(* LS Electric XG5000 project: BURNER110526 *)
(* PLC LSPLC *)
(* module base 0 slot 0: FEnet:XGL-EFMT(B) (Fast Ethernet Module, Electrical Master) *)
(* module base 0 slot 1: Cnet:XGL-C42A/B (Cnet Module(RS-422/485, RS-422/485)) *)
(* module base 0 slot 2: Input Module:XGI-D24A/B (DC 24V Input, 32 Contacts) *)
(* module base 0 slot 3: Input Module:XGI-D24A/B (DC 24V Input, 32 Contacts) *)
(* module base 0 slot 4: Output Module:XGQ-RY2A/B (Relay Output, 16 Contacts (2A, No Varistor/Varistor)) *)
(* module base 0 slot 5: Output Module:XGQ-RY2A/B (Relay Output, 16 Contacts (2A, No Varistor/Varistor)) *)
(* module base 0 slot 6: Analog Output Module:XGF-DC4S (Isolated-type Current Output Type(4 Channels)) *)
(* module base 0 slot 7: Analog Input Module:XGF-AD8A (A/D Voltage/Current Input Type(8 Channels)) *)
(* module base 0 slot 8: Temp. Measuring Module:XGF-RD4A (Temperature Input Type(4 Channels)) *)
VAR_GLOBAL
    GIA_TRI_SV : BOOL;
    _0006_CH0_DATA AT %UW0.6.3 : INT; (* Analog Output Module: CH0 Input *)
    _0006_CH0_OUTEN AT %UX0.6.32 : BOOL; (* Analog Output Module: CH0 Output Enable *)
    _0006_CH1_DATA AT %UW0.6.4 : INT; (* Analog Output Module: CH1 Input *)
    _0006_CH1_OUTEN AT %UX0.6.33 : BOOL; (* Analog Output Module: CH1 Output Enable *)
    _0006_CH2_DATA AT %UW0.6.5 : INT; (* Analog Output Module: CH2 Input *)
    _0006_CH2_OUTEN AT %UX0.6.34 : BOOL; (* Analog Output Module: CH2 Output Enable *)
    _0007_CH0_ACT AT %UX0.7.16 : BOOL; (* Analog Input Module: CH0 Activation Status *)
    _0007_CH0_DATA AT %UW0.7.2 : INT; (* Analog Input Module: CH0 Output *)
    _0007_CH1_ACT AT %UX0.7.17 : BOOL; (* Analog Input Module: CH1 Activation Status *)
    _0007_CH1_DATA AT %UW0.7.3 : INT; (* Analog Input Module: CH1 Output *)
    _0008_CH0_ACT AT %UX0.8.16 : BOOL; (* Temp. Measuring Module: CH0 Activation Status *)
    _0008_CH0_TEMP AT %UW0.8.4 : INT; (* Temp. Measuring Module: CH0 Temp. Data *)
END_VAR

(* Comments on direct variables
%MX98	Burner_Doul
%MX186	HMI_REMOTE
%MX187	HMI_LOCAL
%MX188	HMI_TEX_REMOTE
%MX189	HMI_TEX_LOCAL
%MX192	HMI_REMOTTE
%MX193	HMO_LOACAL
%MW15	DATA_MV_GZ900_ESV
%MW16	DATA_PV_GZ900_ESV
%MW17	DATA_SV_GZ900_ESV
%MW18	DATA_OVER_HTP_ESV
*)

PROGRAM NewProgram (* task: Scan Program *)
VAR
    AIR_CHECK : BOOL;
    AIR_CHECK_OK : BOOL;
    ALARM_AIR_SPEDD : BOOL;
    Alarm_ESV AT %MW5.8 : BOOL;
    ALARM_HIGHT_TEMP : BOOL;
    ALARM_MISS_FIRE : BOOL;
    ALARM_NO1_SHUT : BOOL;
    ALARM_NO2_SHUT : BOOL;
    ALARM_PRESS : BOOL;
    ALARM_SEVOR_HIG : BOOL;
    ALARM_SEVOR_LOW : BOOL;
    BUNER_START : BOOL;
    Burner_Doul AT %MX98 : BOOL;
    burner_Sing AT %MW6.1 : BOOL;
    BUR_START_PER AT %MW1.5 : BOOL; (* BURNER START PERMISSIVE *)
    B_EMG_STOP AT %MW0.0 : BOOL; (* EMEGENCY STOP *)
    B_RESET AT %MW0.1 : BOOL; (* BUTTON RESET *)
    checkk : BOOL;
    CHECK_HIG_SEVOR_OK : BOOL;
    CHECK_NO1_SHUT_OK : BOOL;
    CHECK_NO2_SHUT_OK : BOOL;
    Circulation_Low_Speed_ESV AT %MW5.2 : BOOL;
    Combustion_Air_Fan_Fault_ESV AT %MW4.13 : BOOL;
    Combustion_Air_Fan_Run_ESV AT %MW4.2 : BOOL;
    ECOR_TRIP : BOOL;
    Emergency_Stop_ESV AT %MW5.1 : BOOL;
    FAN_RUN AT %MW0.6 : BOOL; (* LOW CIRCULATION FAN SPEED *)
    FLAMON : BOOL;
    Gas_Leak_Check_Switch_Fault_ESV AT %MW5.4 : BOOL;
    Gas_Leak_PSH_ESV AT %MW4.5 : BOOL;
    Gas_Leak_PSL_ESV AT %MW5.0 : BOOL;
    Gas_Pressure_Hi_ESV AT %MW4.8 : BOOL;
    Gas_Pressure_Low_ESV AT %MW5.3 : BOOL;
    HIGH_GAS_LEAK_PRE AT %MW1.11 : BOOL; (* HIGH GAS LEAK PRESSURE CONTROL SWITCH *)
    HIGH_GAS_PRE AT %MW1.8 : BOOL; (* HIGH GAS PRESSURE *)
    HIGH_LIMIT : BOOL;
    HIGH_SEVOR_CHECK : BOOL;
    Hi_Fire_Limit_Switch_ESV AT %MW4.3 : BOOL;
    Hi_Fire_Limit_Switch_Fault_ESV AT %MW4.12 : BOOL;
    HMI : BOOL;
    HPV_Temp AT %MW507 : INT;
    HPV_Temp1 AT %MW508 : INT;
    INST : TON;
    INST1 : TON;
    INST10 : TON;
    INST11 : TON;
    INST12 : TON;
    INST13 : TON;
    INST14 : TON;
    INST15 : TON;
    INST16 : TON;
    INST17 : TON;
    INST18 : TON;
    INST19 : TON;
    INST2 : TON;
    INST20 : TON;
    INST21 : TON;
    INST22 : TON;
    INST23 : TON;
    INST24 : CTU_INT;
    INST25 : TON;
    INST26 : TON;
    INST27 : TON;
    INST28 : TON;
    INST29 : TON;
    INST3 : TON;
    INST30 : TON;
    INST4 : TON;
    INST5 : TON;
    INST6 : TON;
    INST7 : TON;
    INST8 : TON;
    INST9 : TON;
    LOW_AIR_PRE : BOOL;
    Low_Comb_Air_Fan_Pr_ESV AT %MW4.9 : BOOL;
    LOW_FIRE : BOOL;
    LOW_GAS_LEAK_PRE AT %MW1.10 : BOOL; (* LOW GAS LEAK PRESSURE CONTROL SWITCH *)
    LOW_GAS_PRE AT %MW1.7 : BOOL; (* LOW GAS PRESSURE *)
    LOW_LIMIT : BOOL;
    LOW_LIMIT_CHECK_OK : BOOL;
    Lo_Fire_Limit_Switch_ESV AT %MW4.14 : BOOL;
    Lo_Fire_Limit_Switch_Fault_ESV AT %MW5.7 : BOOL;
    Main_Burner_Miss_Fire_ESV AT %MW5.6 : BOOL;
    MAIN_BURNER_START : BOOL;
    Main_Gas_Shutoff_ESV AT %MW4.15 : BOOL;
    MAIN_PANEL_READY : BOOL;
    Man_Auto_GZ900 AT %MW101 : INT;
    Man_MV_GZ900 AT %MW100 : INT;
    MG : BOOL;
    MG1 AT %MW0.4 : BOOL; (* #1  COMBUSTION FAN RUN *)
    MG2 AT %MW0.5 : BOOL; (* #2  COMBUSTION FAN RUN *)
    MV_GZ900_OUT : INT;
    MƯ20 : WORD;
    mư4 : WORD;
    NO1_ECOR_TRIP AT %MW0.2 : BOOL; (* #1 FAN ECOR TRIP *)
    NO1_FLAME_ON AT %MW1.14 : BOOL; (* #1 BURNER FLAME ON SIGNAL *)
    NO1_HIGH_LIMIT AT %MW1.1 : BOOL; (* #1 HIGH FIRE LIMIT SWITCH *)
    NO1_LOW_AIR_PRE AT %MW1.9 : BOOL; (* #1 LOW COMBUSTION AIR PRESSURE *)
    NO1_LOW_LIMIT AT %MW1.0 : BOOL; (* #1 LOW FIRE LIMIT SWITCH *)
    NO1_SHUT_CHECK : BOOL;
    NO1_SHUT_OFF_SW AT %MW1.13 : BOOL; (* #1 MAIN SHUT_OFF VAVLE CLOSED LIMIT SWITCH *)
    NO2_ECOR_TRIP AT %MW0.3 : BOOL; (* #2 FAN ECOR TRIP *)
    NO2_FLAME_ON AT %MW1.15 : BOOL; (* #2 BURNER FLAME ON SIGNAL *)
    NO2_HIGH_LIMIT AT %MW1.3 : BOOL; (* #2 HIGH FIRE LIMIT SWITCH *)
    NO2_LOW_AIR_PRE AT %MW1.12 : BOOL; (* #2 LOW COMBUSTION AIR PRESSURE *)
    NO2_LOW_LIMIT AT %MW1.2 : BOOL; (* #2 LOW FIRE LIMIT SWITCH *)
    NO2_SHUT_CHECK : BOOL;
    NO_READY : BOOL;
    O502 AT %MW3.0 : BOOL; (* BURNER LOAD UP *)
    O503 AT %MW3.1 : BOOL; (* LOW CIRCULATION FAN SPEED *)
    O504 AT %MW3.2 : BOOL; (* BURNER START *)
    O505 AT %MW3.3 : BOOL;
    O506 AT %MW3.4 : BOOL; (* HIGH TEMPERATURE *)
    O507 AT %MW3.5 : BOOL; (* MISS FIRE *)
    O508 AT %MW3.6 : BOOL; (* HIGH GAS PRESSURE *)
    O509 AT %MW3.7 : BOOL; (* LOW GAS PRESSURE *)
    O510 AT %MW3.8 : BOOL; (* GAS LEAK FAULT *)
    O511 AT %MW3.9 : BOOL; (* PURGE START *)
    O512 AT %MW3.10 : BOOL; (* PURGE END *)
    O513 AT %MW3.11 : BOOL; (* NO 1 LOW COMBUSTION FAN PRESSURE *)
    O514 AT %MW3.12 : BOOL; (* NO 1 LOW COMBUSTION FAN RUNNING *)
    O515 AT %MW3.13 : BOOL; (* NO 2 LOW COMBUSTION FAN PRESSURE *)
    O516 AT %MW3.14 : BOOL; (* NO 2 LOW COMBUSTION FAN RUNNING *)
    O517 AT %MW3.15 : BOOL;
    O518 AT %MW2.14 : BOOL; (* NO.01 COMBUSTION FAN ECOR TRIP *)
    O519 AT %MW2.15 : BOOL; (* NO.02 COMBUSTION FAN ECOR TRIP *)
    Operation_Remote_Mode_ESV AT %MW4.6 : BOOL;
    Pilot_Burner_Miss_Fire_ESV AT %MW4.11 : BOOL;
    PILOT_INR : BOOL;
    Pilot_Valve_ESV AT %MW4.4 : BOOL;
    PV_GZ900 AT %MW103 : INT;
    PV_GZ900_OUT : INT;
    Ready_ESV AT %MW4.0 : BOOL;
    Remote_ESV AT %MW4.1 : BOOL;
    RE_RESET AT %MW1.6 : BOOL; (* REMOTE RESET *)
    RE_START AT %MW1.4 : BOOL; (* REMOTE START *)
    RMV_GZ900 AT %MW104 : INT;
    START : BOOL;
    STOP AT %MW6.0 : BOOL;
    STOP_BURNER : BOOL;
    SV_GZ900 AT %MW102 : INT;
    SV_THIC_Data AT %MW506 : INT;
    SV_TIC_Data AT %MW505 : INT;
    temp1 : INT;
    temp2 : INT;
    Temp_high_ESV AT %MW4.7 : BOOL;
    WMV_GZ900 AT %MW504 : INT;
    WPV AT %MW520 : INT;
    WPV_GZ900 AT %MW503 : INT;
    _1ST_Valve_Gas_leak_ESV AT %MW4.10 : BOOL;
    _2ND_Valve_Gas_leak_ESV AT %MW5.5 : BOOL;
END_VAR
VAR_EXTERNAL
    _0006_CH0_DATA : INT; (* AT %UW0.6.3 *) (* Analog Output Module: CH0 Input *)
    _0006_CH0_OUTEN : BOOL; (* AT %UX0.6.32 *) (* Analog Output Module: CH0 Output Enable *)
    _0006_CH1_DATA : INT; (* AT %UW0.6.4 *) (* Analog Output Module: CH1 Input *)
    _0006_CH1_OUTEN : BOOL; (* AT %UX0.6.33 *) (* Analog Output Module: CH1 Output Enable *)
    _0006_CH2_DATA : INT; (* AT %UW0.6.5 *) (* Analog Output Module: CH2 Input *)
    _0006_CH2_OUTEN : BOOL; (* AT %UX0.6.34 *) (* Analog Output Module: CH2 Output Enable *)
    _0007_CH0_ACT : BOOL; (* AT %UX0.7.16 *) (* Analog Input Module: CH0 Activation Status *)
    _0007_CH0_DATA : INT; (* AT %UW0.7.2 *) (* Analog Input Module: CH0 Output *)
    _0007_CH1_ACT : BOOL; (* AT %UX0.7.17 *) (* Analog Input Module: CH1 Activation Status *)
    _0007_CH1_DATA : INT; (* AT %UW0.7.3 *) (* Analog Input Module: CH1 Output *)
    _0008_CH0_ACT : BOOL; (* AT %UX0.8.16 *) (* Temp. Measuring Module: CH0 Activation Status *)
    _0008_CH0_TEMP : INT; (* AT %UW0.8.4 *) (* Temp. Measuring Module: CH0 Temp. Data *)
END_VAR
VAR
    _e1 : R_TRIG;
    _e2 : R_TRIG;
    _e3 : F_TRIG;
    _e4 : R_TRIG;
    _e5 : R_TRIG;
    _p6 : BOOL;
    _p7 : BOOL;
    _e8 : R_TRIG;
    _e9 : R_TRIG;
    _p10 : BOOL;
    _p11 : BOOL;
    _p12 : BOOL;
    _p13 : BOOL;
    _p14 : BOOL;
    _p15 : BOOL;
    _p16 : BOOL;
    _p17 : BOOL;
    _p18 : BOOL;
    _t19 : BOOL;
    _t20 : BOOL;
END_VAR

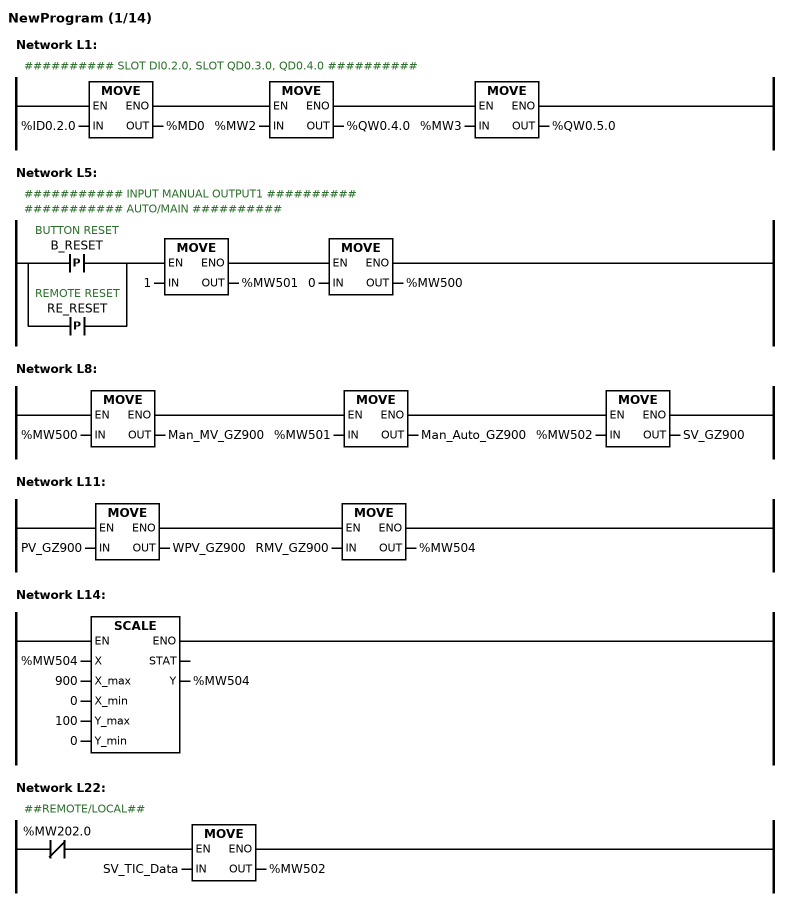
(* ########## SLOT DI0.2.0, SLOT QD0.3.0, QD0.4.0 ########## *)
(* Rung L1 *)
%MD0 := %ID0.2.0;
%QW0.4.0 := %MW2;
%QW0.5.0 := %MW3;
(* ########### INPUT MANUAL OUTPUT1 ########## / ########### AUTO/MAIN ########## *)
(* Rung L5 *)
_e1(CLK := B_RESET);
_e2(CLK := RE_RESET);
IF _e1.Q OR _e2.Q THEN
    %MW501 := 1;
    %MW500 := 0;
END_IF;
(* Rung L8 *)
Man_MV_GZ900 := %MW500;
Man_Auto_GZ900 := %MW501;
SV_GZ900 := %MW502;
(* Rung L11 *)
WPV_GZ900 := PV_GZ900;
%MW504 := RMV_GZ900;
(* Rung L14 *)
SCALE(X := %MW504, X_max := 900, X_min := 0, Y_max := 100, Y_min := 0, Y => %MW504);
(* ##REMOTE/LOCAL## *)
(* Rung L22 *)
IF NOT %MW202.0 THEN %MW502 := SV_TIC_Data; END_IF;

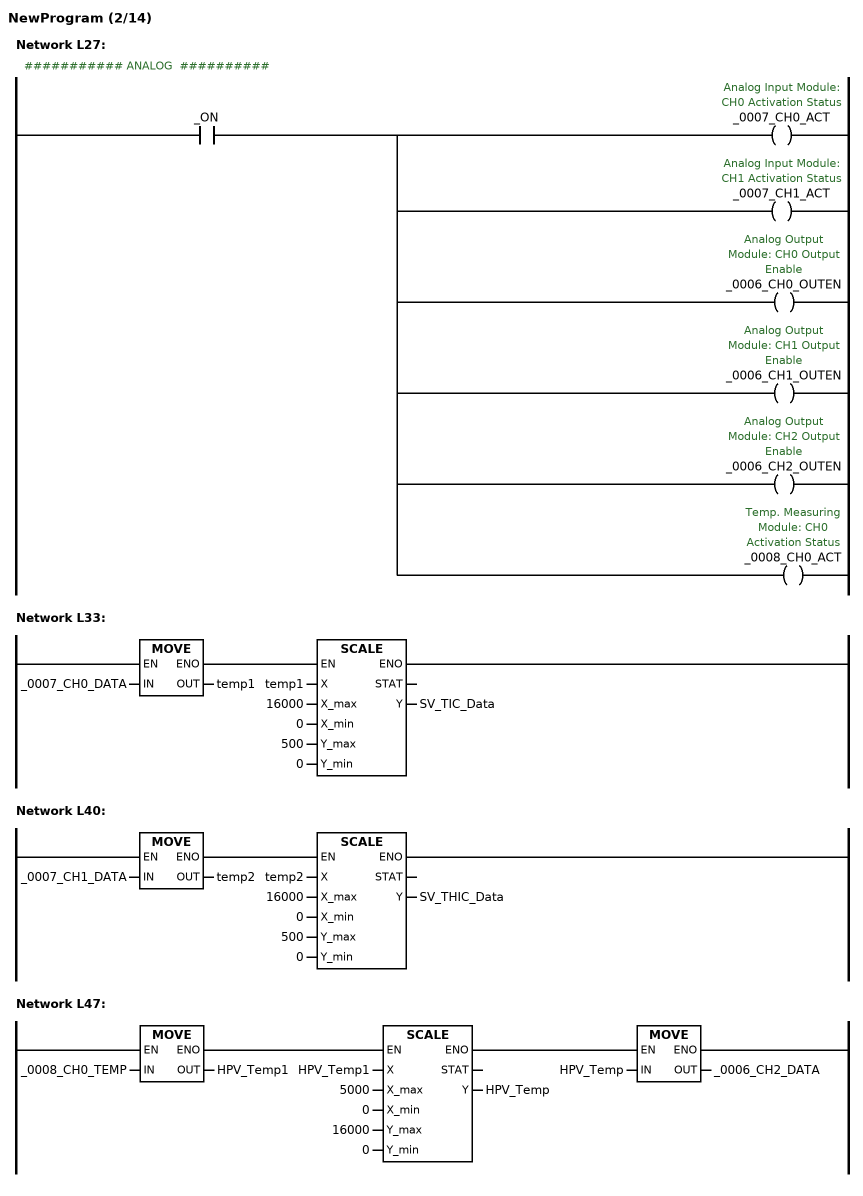
(* ########### ANALOG  ########## *)
(* Rung L27 *)
_0007_CH0_ACT := _ON;
_0007_CH1_ACT := _ON;
_0006_CH0_OUTEN := _ON;
_0006_CH1_OUTEN := _ON;
_0006_CH2_OUTEN := _ON;
_0008_CH0_ACT := _ON;
(* Rung L33 *)
temp1 := _0007_CH0_DATA;
SCALE(X := temp1, X_max := 16000, X_min := 0, Y_max := 500, Y_min := 0, Y => SV_TIC_Data);
(* Rung L40 *)
temp2 := _0007_CH1_DATA;
SCALE(X := temp2, X_max := 16000, X_min := 0, Y_max := 500, Y_min := 0, Y => SV_THIC_Data);
(* Rung L47 *)
HPV_Temp1 := _0008_CH0_TEMP;
SCALE(X := HPV_Temp1, X_max := 5000, X_min := 0, Y_max := 16000, Y_min := 0, Y => HPV_Temp);
_0006_CH2_DATA := HPV_Temp;

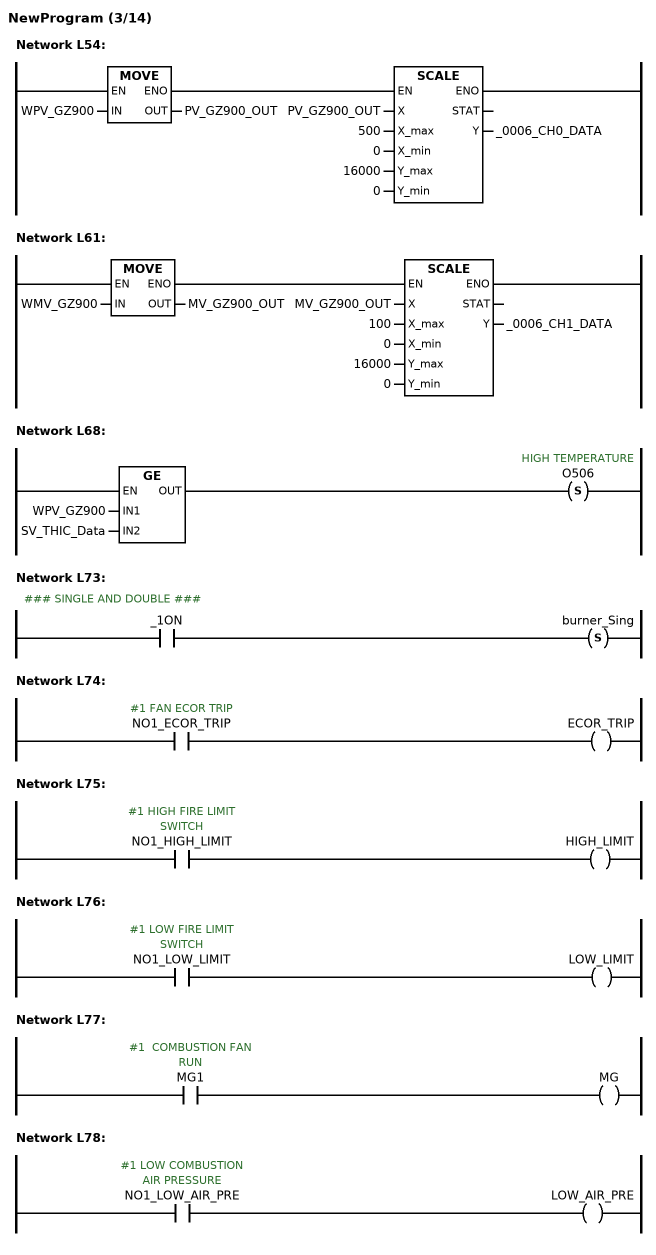
(* Rung L54 *)
PV_GZ900_OUT := WPV_GZ900;
SCALE(X := PV_GZ900_OUT, X_max := 500, X_min := 0, Y_max := 16000, Y_min := 0, Y => _0006_CH0_DATA);
(* Rung L61 *)
MV_GZ900_OUT := WMV_GZ900;
SCALE(X := MV_GZ900_OUT, X_max := 100, X_min := 0, Y_max := 16000, Y_min := 0, Y => _0006_CH1_DATA);
(* Rung L68 *)
IF WPV_GZ900 >= SV_THIC_Data THEN O506 := TRUE; END_IF;
(* ### SINGLE AND DOUBLE ### *)
(* Rung L73 *)
IF _1ON THEN burner_Sing := TRUE; END_IF;
(* Rung L74 *)
ECOR_TRIP := NO1_ECOR_TRIP;
(* Rung L75 *)
HIGH_LIMIT := NO1_HIGH_LIMIT;
(* Rung L76 *)
LOW_LIMIT := NO1_LOW_LIMIT;
(* Rung L77 *)
MG := MG1;
(* Rung L78 *)
LOW_AIR_PRE := NO1_LOW_AIR_PRE;

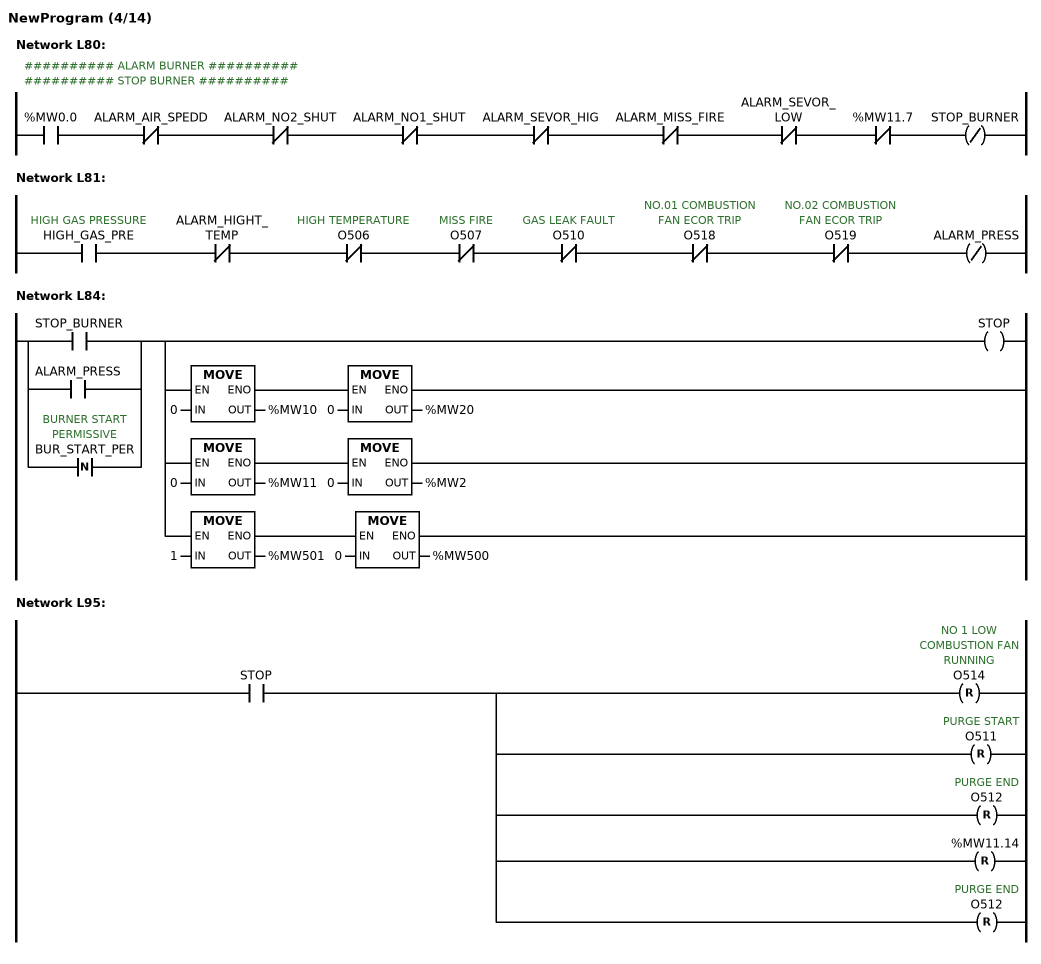
(* ########## ALARM BURNER ########## / ########## STOP BURNER ########## *)
(* Rung L80 *)
STOP_BURNER := NOT (%MW0.0 AND NOT ALARM_AIR_SPEDD AND NOT ALARM_NO2_SHUT AND NOT ALARM_NO1_SHUT AND NOT ALARM_SEVOR_HIG AND NOT ALARM_MISS_FIRE AND NOT ALARM_SEVOR_LOW AND NOT %MW11.7);
(* Rung L81 *)
ALARM_PRESS := NOT (HIGH_GAS_PRE AND NOT ALARM_HIGHT_TEMP AND NOT O506 AND NOT O507 AND NOT O510 AND NOT O518 AND NOT O519);
(* Rung L84 *)
_e3(CLK := BUR_START_PER);
STOP := STOP_BURNER OR ALARM_PRESS OR _e3.Q;
IF STOP_BURNER OR ALARM_PRESS OR _e3.Q THEN
    %MW10 := 0;
    %MW20 := 0;
    %MW11 := 0;
    %MW2 := 0;
    %MW501 := 1;
    %MW500 := 0;
END_IF;
(* Rung L95 *)
IF STOP THEN
    O514 := FALSE;
    O511 := FALSE;
    O512 := FALSE;
    %MW11.14 := FALSE;
    O512 := FALSE;
END_IF;

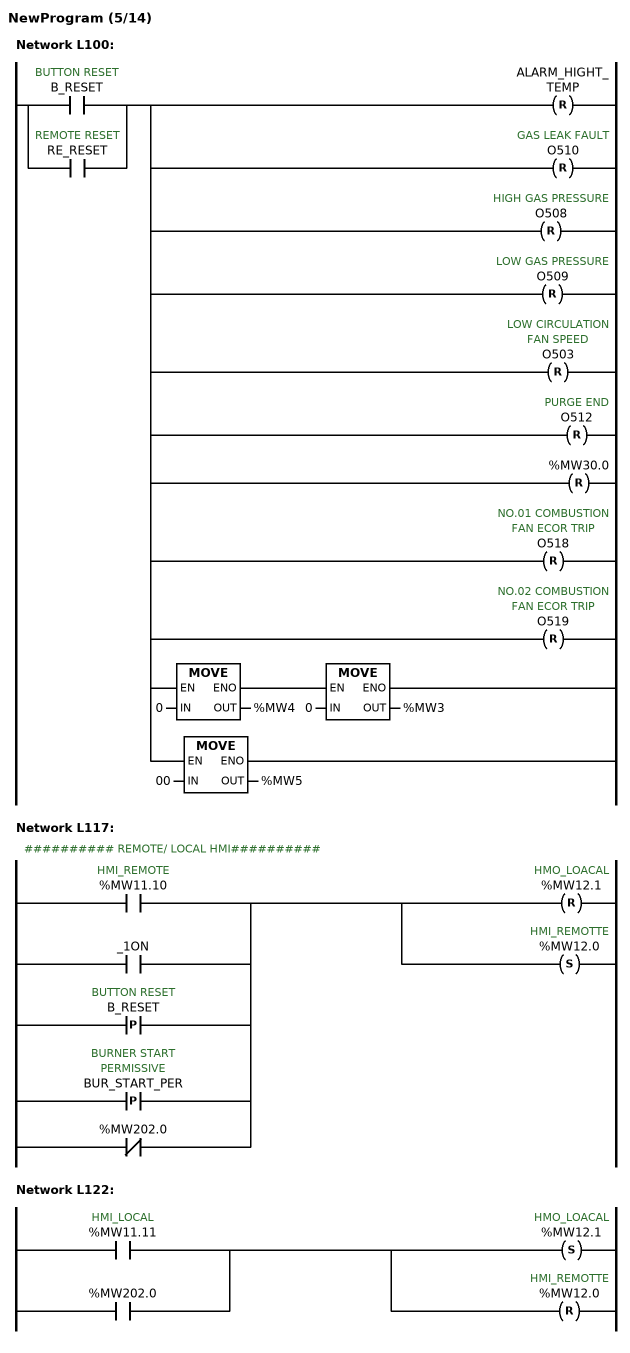
(* Rung L100 *)
IF B_RESET OR RE_RESET THEN
    ALARM_HIGHT_TEMP := FALSE;
    O510 := FALSE;
    O508 := FALSE;
    O509 := FALSE;
    O503 := FALSE;
    O512 := FALSE;
    %MW30.0 := FALSE;
    O518 := FALSE;
    O519 := FALSE;
    %MW4 := 0;
    %MW3 := 0;
    %MW5 := 00;
END_IF;
(* ########## REMOTE/ LOCAL HMI########## *)
(* Rung L117 *)
_e4(CLK := B_RESET);
_e5(CLK := BUR_START_PER);
_p6 := %MW11.10 OR _1ON OR _e4.Q OR _e5.Q OR NOT %MW202.0;
IF _p6 THEN
    %MW12.1 := FALSE;
    %MW12.0 := TRUE;
END_IF;
(* Rung L122 *)
IF %MW11.11 OR %MW202.0 THEN
    %MW12.1 := TRUE;
    %MW12.0 := FALSE;
END_IF;

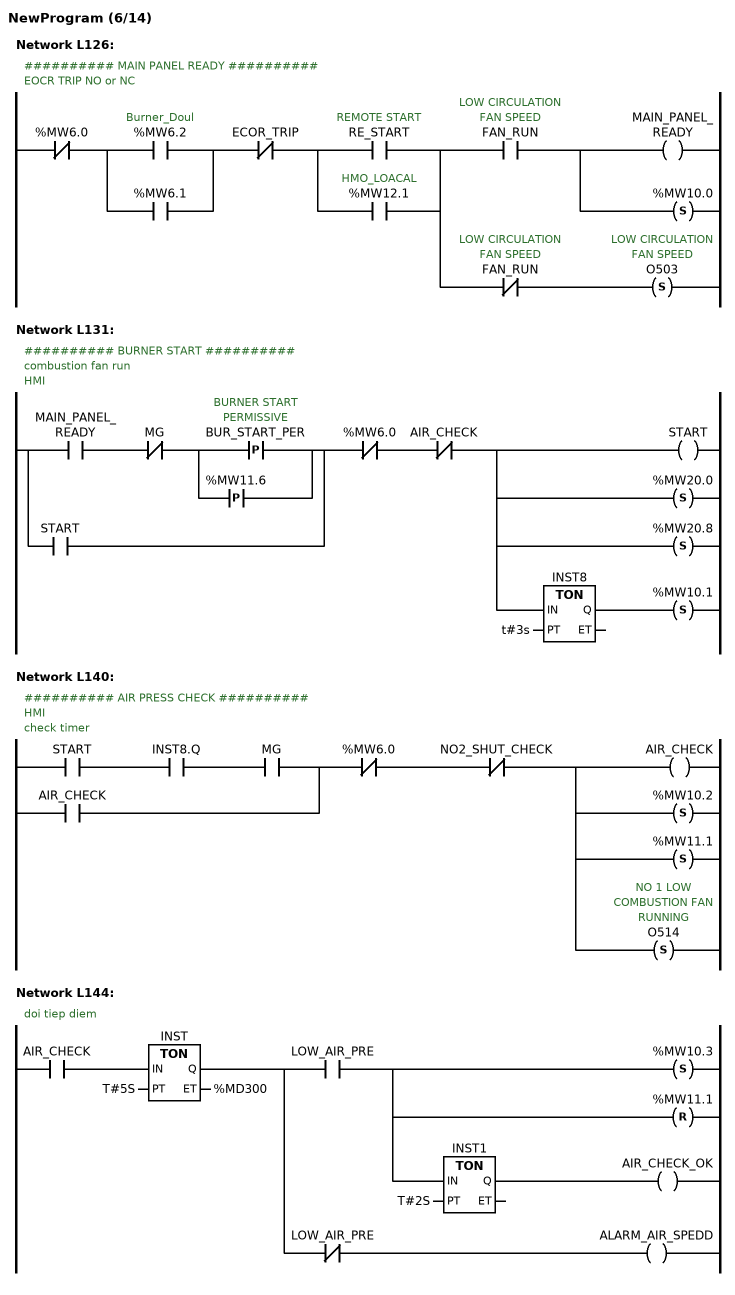
(* ########## MAIN PANEL READY ########## *)
(* Rung L126 *)
_p7 := NOT %MW6.0 AND (%MW6.2 OR %MW6.1) AND NOT ECOR_TRIP AND (RE_START OR %MW12.1);
MAIN_PANEL_READY := _p7 AND FAN_RUN;
IF _p7 AND FAN_RUN THEN %MW10.0 := TRUE; END_IF;
IF _p7 AND NOT FAN_RUN THEN O503 := TRUE; END_IF;
(* EOCR TRIP NO or NC *)
(* ########## BURNER START ########## *)
(* Rung L131 *)
_e8(CLK := BUR_START_PER);
_e9(CLK := %MW11.6);
_p10 := ((MAIN_PANEL_READY AND NOT MG AND (_e8.Q OR _e9.Q)) OR START) AND NOT %MW6.0 AND NOT AIR_CHECK;
START := _p10;
IF _p10 THEN
    %MW20.0 := TRUE;
    %MW20.8 := TRUE;
END_IF;
INST8(IN := _p10, PT := t#3s);
IF INST8.Q THEN %MW10.1 := TRUE; END_IF;
(* combustion fan run *)
(* HMI *)
(* ########## AIR PRESS CHECK ########## *)
(* Rung L140 *)
_p11 := ((START AND INST8.Q AND MG) OR AIR_CHECK) AND NOT %MW6.0 AND NOT NO2_SHUT_CHECK;
AIR_CHECK := _p11;
IF _p11 THEN
    %MW10.2 := TRUE;
    %MW11.1 := TRUE;
    O514 := TRUE;
END_IF;
(* HMI *)
(* check timer *)
(* Rung L144 *)
INST(IN := AIR_CHECK, PT := T#5S, ET => %MD300);
IF INST.Q AND LOW_AIR_PRE THEN
    %MW10.3 := TRUE;
    %MW11.1 := FALSE;
END_IF;
INST1(IN := INST.Q AND LOW_AIR_PRE, PT := T#2S);
AIR_CHECK_OK := INST1.Q;
ALARM_AIR_SPEDD := INST.Q AND NOT LOW_AIR_PRE;
(* doi tiep diem *)

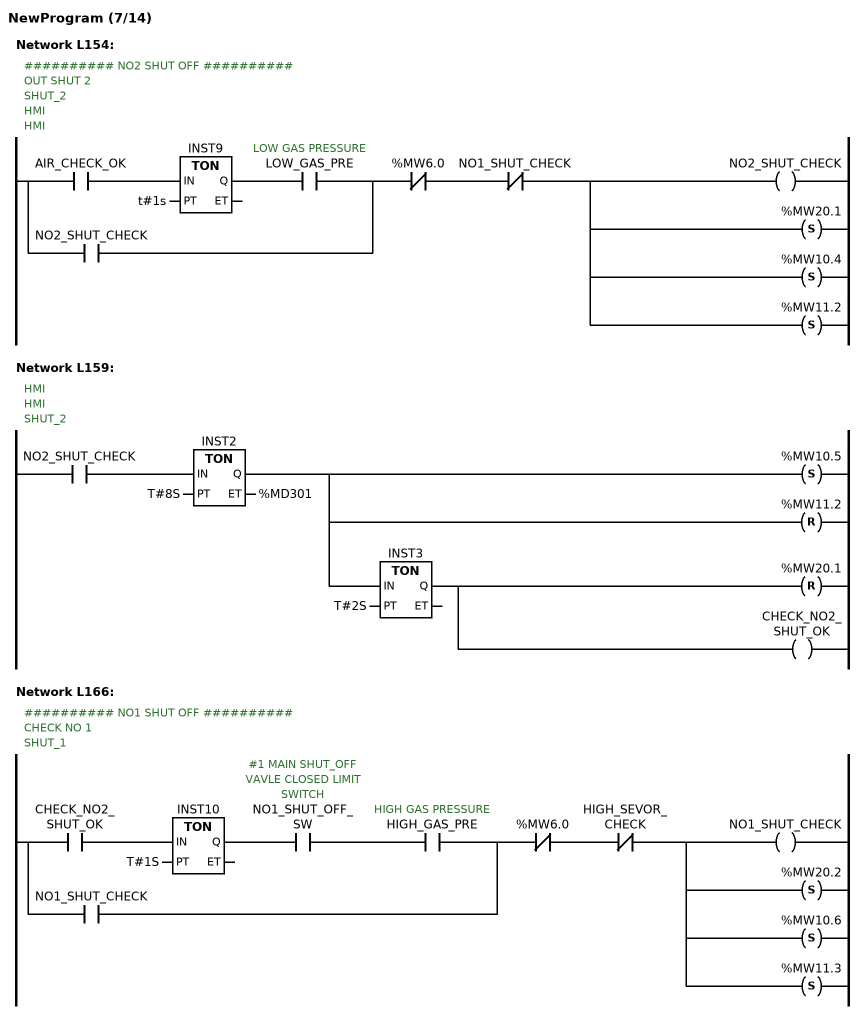
(* ########## NO2 SHUT OFF ########## *)
(* Rung L154 *)
INST9(IN := AIR_CHECK_OK, PT := t#1s);
_p12 := ((INST9.Q AND LOW_GAS_PRE) OR NO2_SHUT_CHECK) AND NOT %MW6.0 AND NOT NO1_SHUT_CHECK;
NO2_SHUT_CHECK := _p12;
IF _p12 THEN
    %MW20.1 := TRUE;
    %MW10.4 := TRUE;
    %MW11.2 := TRUE;
END_IF;
(* OUT SHUT 2 *)
(* SHUT_2 *)
(* HMI *)
(* HMI *)
(* Rung L159 *)
INST2(IN := NO2_SHUT_CHECK, PT := T#8S, ET => %MD301);
IF INST2.Q THEN
    %MW10.5 := TRUE;
    %MW11.2 := FALSE;
END_IF;
INST3(IN := INST2.Q, PT := T#2S);
IF INST3.Q THEN %MW20.1 := FALSE; END_IF;
CHECK_NO2_SHUT_OK := INST3.Q;
(* HMI *)
(* HMI *)
(* SHUT_2 *)
(* ########## NO1 SHUT OFF ########## *)
(* Rung L166 *)
INST10(IN := CHECK_NO2_SHUT_OK, PT := T#1S);
_p13 := ((INST10.Q AND NO1_SHUT_OFF_SW AND HIGH_GAS_PRE) OR NO1_SHUT_CHECK) AND NOT %MW6.0 AND NOT HIGH_SEVOR_CHECK;
NO1_SHUT_CHECK := _p13;
IF _p13 THEN
    %MW20.2 := TRUE;
    %MW10.6 := TRUE;
    %MW11.3 := TRUE;
END_IF;
(* CHECK NO 1 *)
(* SHUT_1 *)

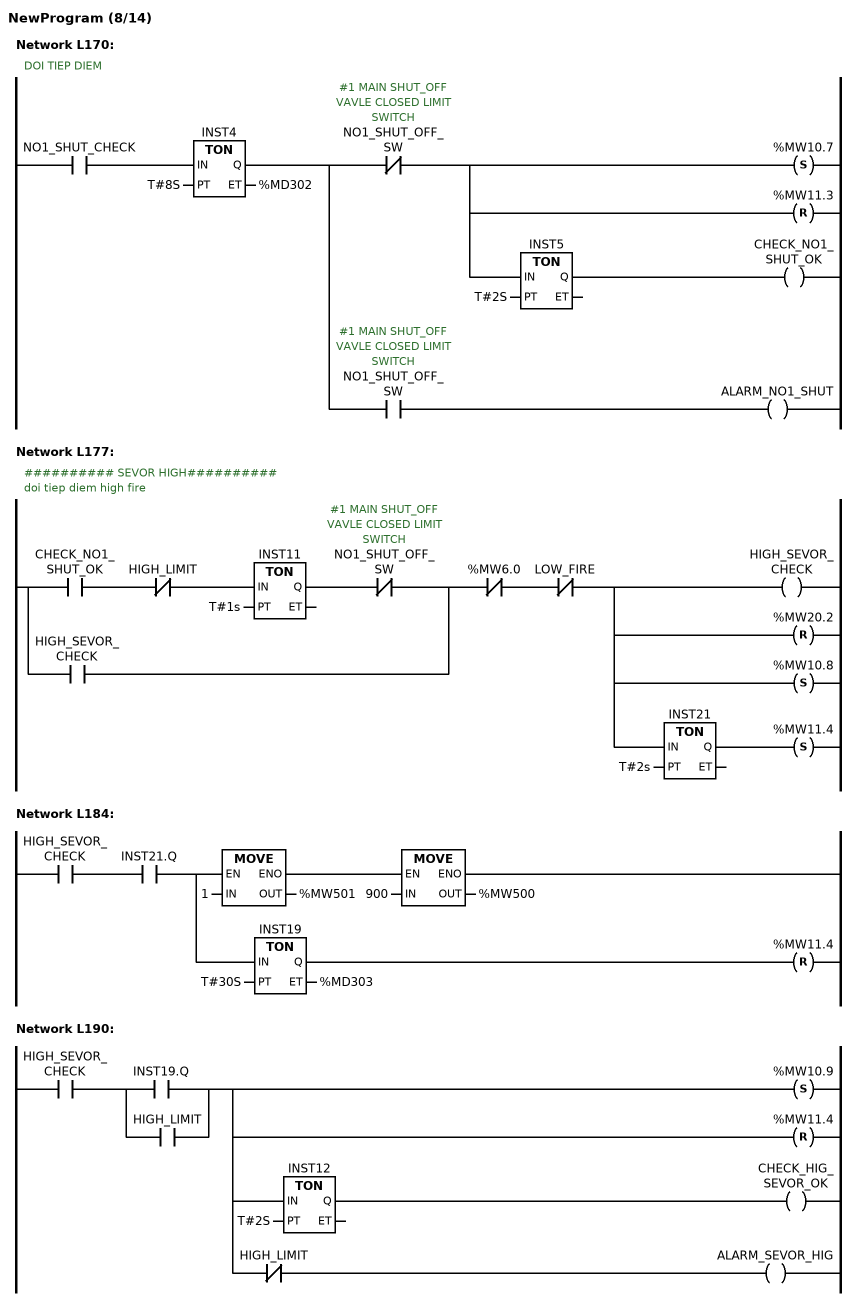
(* Rung L170 *)
INST4(IN := NO1_SHUT_CHECK, PT := T#8S, ET => %MD302);
IF INST4.Q AND NOT NO1_SHUT_OFF_SW THEN
    %MW10.7 := TRUE;
    %MW11.3 := FALSE;
END_IF;
INST5(IN := INST4.Q AND NOT NO1_SHUT_OFF_SW, PT := T#2S);
CHECK_NO1_SHUT_OK := INST5.Q;
ALARM_NO1_SHUT := INST4.Q AND NO1_SHUT_OFF_SW;
(* DOI TIEP DIEM *)
(* ########## SEVOR HIGH########## *)
(* Rung L177 *)
INST11(IN := CHECK_NO1_SHUT_OK AND NOT HIGH_LIMIT, PT := T#1s);
_p14 := ((INST11.Q AND NOT NO1_SHUT_OFF_SW) OR HIGH_SEVOR_CHECK) AND NOT %MW6.0 AND NOT LOW_FIRE;
HIGH_SEVOR_CHECK := _p14;
IF _p14 THEN
    %MW20.2 := FALSE;
    %MW10.8 := TRUE;
END_IF;
INST21(IN := _p14, PT := T#2s);
IF INST21.Q THEN %MW11.4 := TRUE; END_IF;
(* doi tiep diem high fire *)
(* Rung L184 *)
IF HIGH_SEVOR_CHECK AND INST21.Q THEN
    %MW501 := 1;
    %MW500 := 900;
END_IF;
INST19(IN := HIGH_SEVOR_CHECK AND INST21.Q, PT := T#30S, ET => %MD303);
IF INST19.Q THEN %MW11.4 := FALSE; END_IF;
(* Rung L190 *)
IF HIGH_SEVOR_CHECK AND (INST19.Q OR HIGH_LIMIT) THEN
    %MW10.9 := TRUE;
    %MW11.4 := FALSE;
END_IF;
INST12(IN := HIGH_SEVOR_CHECK AND (INST19.Q OR HIGH_LIMIT), PT := T#2S);
CHECK_HIG_SEVOR_OK := INST12.Q;
ALARM_SEVOR_HIG := HIGH_SEVOR_CHECK AND (INST19.Q OR HIGH_LIMIT) AND NOT HIGH_LIMIT;
(*  *)

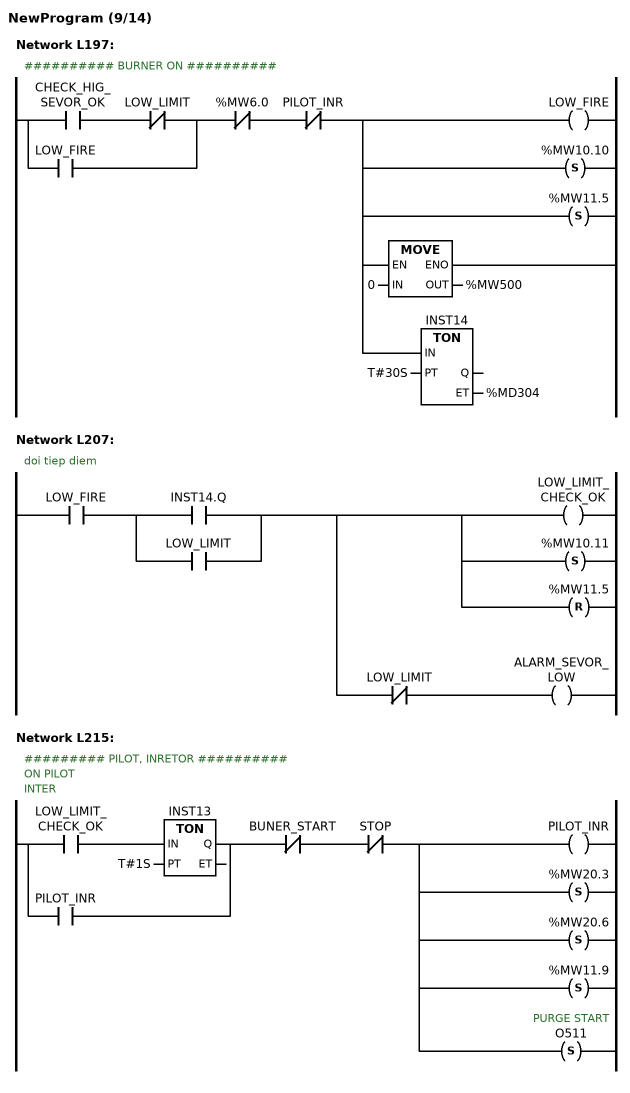
(* ########## BURNER ON ########## *)
(* Rung L197 *)
_p15 := ((CHECK_HIG_SEVOR_OK AND NOT LOW_LIMIT) OR LOW_FIRE) AND NOT %MW6.0 AND NOT PILOT_INR;
LOW_FIRE := _p15;
IF _p15 THEN
    %MW10.10 := TRUE;
    %MW11.5 := TRUE;
    %MW500 := 0;
END_IF;
INST14(IN := _p15, PT := T#30S, ET => %MD304);
(* Rung L207 *)
LOW_LIMIT_CHECK_OK := LOW_FIRE AND (INST14.Q OR LOW_LIMIT);
IF LOW_FIRE AND (INST14.Q OR LOW_LIMIT) THEN
    %MW10.11 := TRUE;
    %MW11.5 := FALSE;
END_IF;
ALARM_SEVOR_LOW := LOW_FIRE AND (INST14.Q OR LOW_LIMIT) AND NOT LOW_LIMIT;
(* doi tiep diem *)
(* ######### PILOT, INRETOR ########## *)
(* Rung L215 *)
INST13(IN := LOW_LIMIT_CHECK_OK, PT := T#1S);
_p16 := (INST13.Q OR PILOT_INR) AND NOT BUNER_START AND NOT STOP;
PILOT_INR := _p16;
IF _p16 THEN
    %MW20.3 := TRUE;
    %MW20.6 := TRUE;
    %MW11.9 := TRUE;
    O511 := TRUE;
END_IF;
(* ON PILOT *)
(* INTER *)

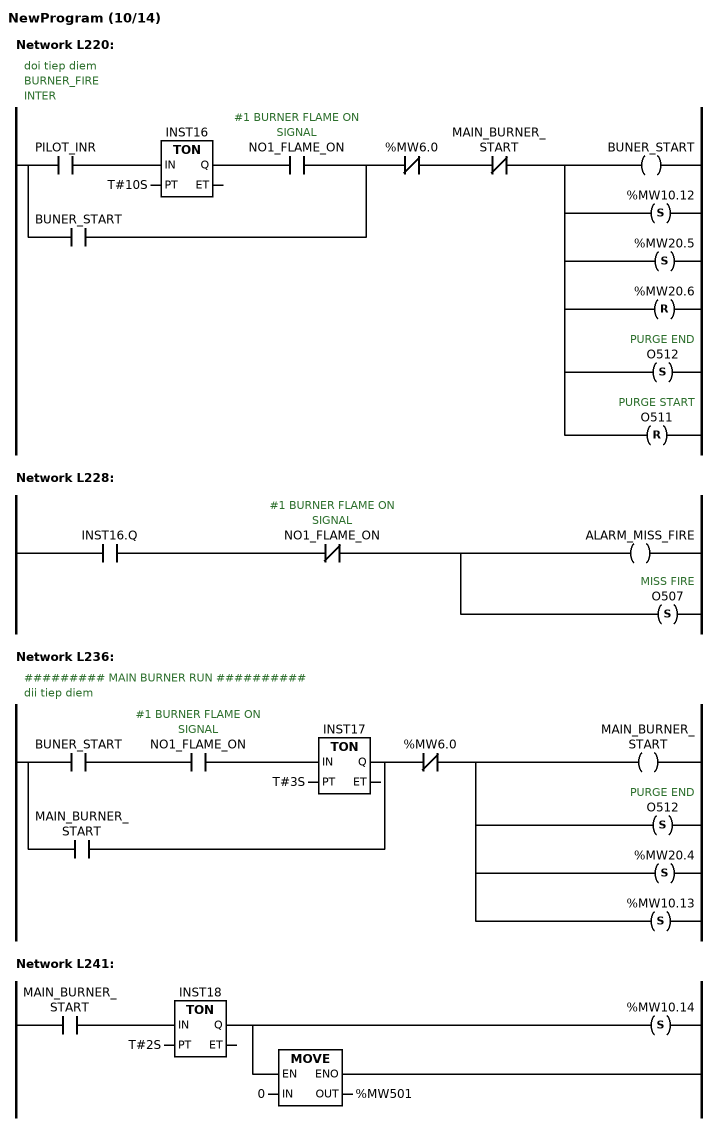
(* Rung L220 *)
INST16(IN := PILOT_INR, PT := T#10S);
_p17 := ((INST16.Q AND NO1_FLAME_ON) OR BUNER_START) AND NOT %MW6.0 AND NOT MAIN_BURNER_START;
BUNER_START := _p17;
IF _p17 THEN
    %MW10.12 := TRUE;
    %MW20.5 := TRUE;
    %MW20.6 := FALSE;
    O512 := TRUE;
    O511 := FALSE;
END_IF;
(* doi tiep diem *)
(* BURNER_FIRE *)
(* INTER *)
(* Rung L228 *)
ALARM_MISS_FIRE := INST16.Q AND NOT NO1_FLAME_ON;
IF INST16.Q AND NOT NO1_FLAME_ON THEN O507 := TRUE; END_IF;
(* ######### MAIN BURNER RUN ########## *)
(* Rung L236 *)
INST17(IN := BUNER_START AND NO1_FLAME_ON, PT := T#3S);
_p18 := (INST17.Q OR MAIN_BURNER_START) AND NOT %MW6.0;
MAIN_BURNER_START := _p18;
IF _p18 THEN
    O512 := TRUE;
    %MW20.4 := TRUE;
    %MW10.13 := TRUE;
END_IF;
(* dii tiep diem *)
(* Rung L241 *)
INST18(IN := MAIN_BURNER_START, PT := T#2S);
IF INST18.Q THEN
    %MW10.14 := TRUE;
    %MW501 := 0;
END_IF;

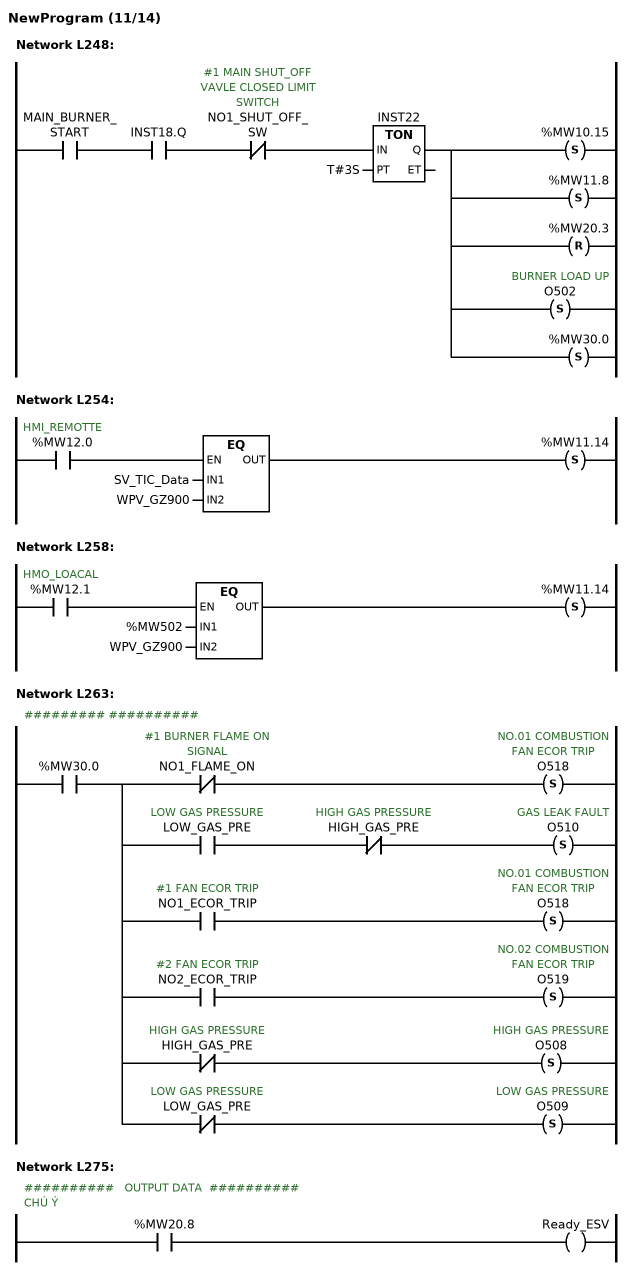
(* Rung L248 *)
INST22(IN := MAIN_BURNER_START AND INST18.Q AND NOT NO1_SHUT_OFF_SW, PT := T#3S);
IF INST22.Q THEN
    %MW10.15 := TRUE;
    %MW11.8 := TRUE;
    %MW20.3 := FALSE;
    O502 := TRUE;
    %MW30.0 := TRUE;
END_IF;
(* Rung L254 *)
IF %MW12.0 THEN _t19 := SV_TIC_Data = WPV_GZ900; END_IF;
IF _t19 THEN %MW11.14 := TRUE; END_IF;
(* Rung L258 *)
IF %MW12.1 THEN _t20 := %MW502 = WPV_GZ900; END_IF;
IF _t20 THEN %MW11.14 := TRUE; END_IF;
(* ######### ########## *)
(* Rung L263 *)
IF %MW30.0 AND NOT NO1_FLAME_ON THEN O518 := TRUE; END_IF;
IF %MW30.0 AND LOW_GAS_PRE AND NOT HIGH_GAS_PRE THEN O510 := TRUE; END_IF;
IF %MW30.0 AND NO1_ECOR_TRIP THEN O518 := TRUE; END_IF;
IF %MW30.0 AND NO2_ECOR_TRIP THEN O519 := TRUE; END_IF;
IF %MW30.0 AND NOT HIGH_GAS_PRE THEN O508 := TRUE; END_IF;
IF %MW30.0 AND NOT LOW_GAS_PRE THEN O509 := TRUE; END_IF;
(* ##########   OUTPUT DATA  ########## *)
(* Rung L275 *)
Ready_ESV := %MW20.8;
(* CHÚ Ý *)

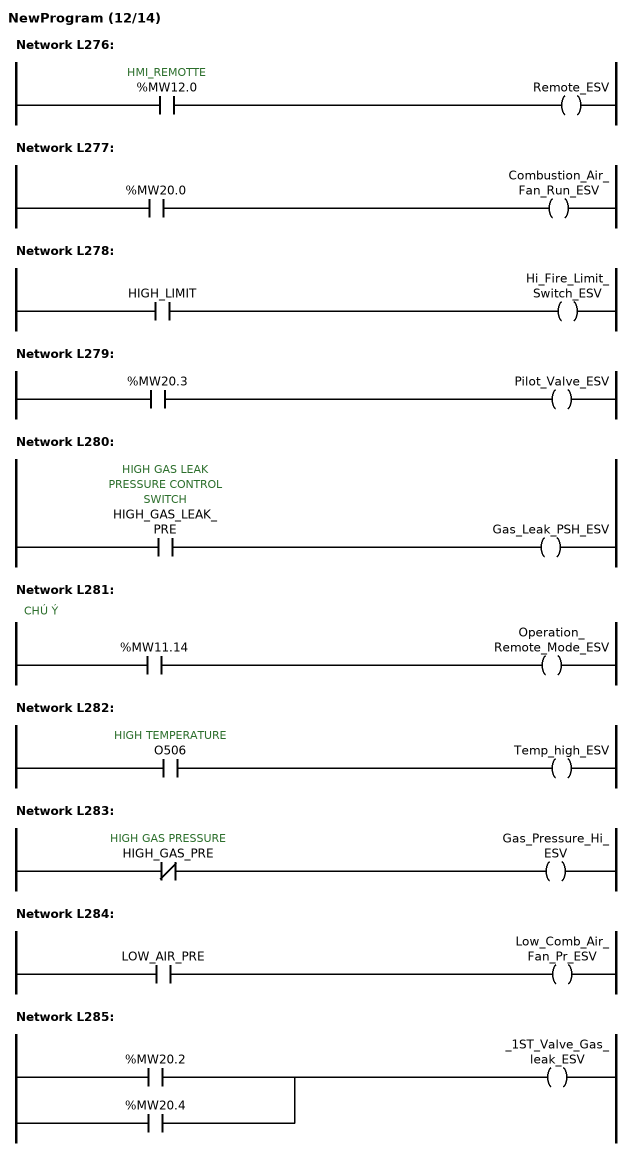
(* Rung L276 *)
Remote_ESV := %MW12.0;
(* Rung L277 *)
Combustion_Air_Fan_Run_ESV := %MW20.0;
(* Rung L278 *)
Hi_Fire_Limit_Switch_ESV := HIGH_LIMIT;
(* Rung L279 *)
Pilot_Valve_ESV := %MW20.3;
(* Rung L280 *)
Gas_Leak_PSH_ESV := HIGH_GAS_LEAK_PRE;
(* Rung L281 *)
Operation_Remote_Mode_ESV := %MW11.14;
(* CHÚ Ý *)
(* Rung L282 *)
Temp_high_ESV := O506;
(* Rung L283 *)
Gas_Pressure_Hi_ESV := NOT HIGH_GAS_PRE;
(* Rung L284 *)
Low_Comb_Air_Fan_Pr_ESV := LOW_AIR_PRE;
(* Rung L285 *)
_1ST_Valve_Gas_leak_ESV := %MW20.2 OR %MW20.4;

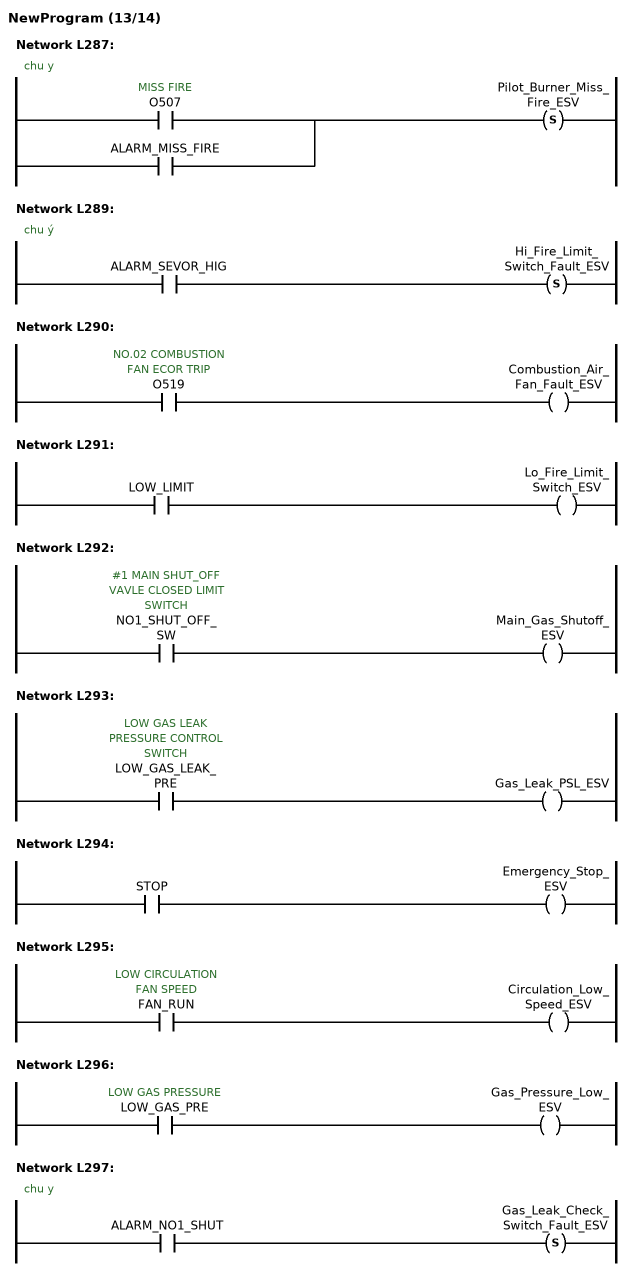
(* Rung L287 *)
IF O507 OR ALARM_MISS_FIRE THEN Pilot_Burner_Miss_Fire_ESV := TRUE; END_IF;
(* chu y *)
(* Rung L289 *)
IF ALARM_SEVOR_HIG THEN Hi_Fire_Limit_Switch_Fault_ESV := TRUE; END_IF;
(* chu ý *)
(* Rung L290 *)
Combustion_Air_Fan_Fault_ESV := O519;
(* Rung L291 *)
Lo_Fire_Limit_Switch_ESV := LOW_LIMIT;
(* Rung L292 *)
Main_Gas_Shutoff_ESV := NO1_SHUT_OFF_SW;
(* Rung L293 *)
Gas_Leak_PSL_ESV := LOW_GAS_LEAK_PRE;
(* Rung L294 *)
Emergency_Stop_ESV := STOP;
(* Rung L295 *)
Circulation_Low_Speed_ESV := FAN_RUN;
(* Rung L296 *)
Gas_Pressure_Low_ESV := LOW_GAS_PRE;
(* Rung L297 *)
IF ALARM_NO1_SHUT THEN Gas_Leak_Check_Switch_Fault_ESV := TRUE; END_IF;
(* chu y *)

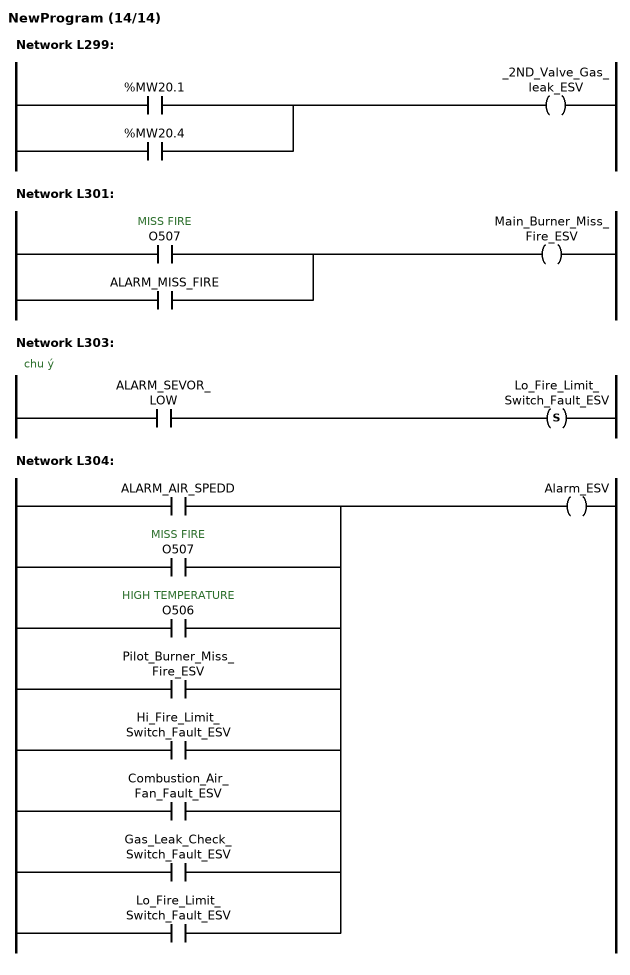
(* Rung L299 *)
_2ND_Valve_Gas_leak_ESV := %MW20.1 OR %MW20.4;
(* Rung L301 *)
Main_Burner_Miss_Fire_ESV := O507 OR ALARM_MISS_FIRE;
(* Rung L303 *)
IF ALARM_SEVOR_LOW THEN Lo_Fire_Limit_Switch_Fault_ESV := TRUE; END_IF;
(* chu ý *)
(* Rung L304 *)
Alarm_ESV := ALARM_AIR_SPEDD OR O507 OR O506 OR Pilot_Burner_Miss_Fire_ESV OR Hi_Fire_Limit_Switch_Fault_ESV OR Combustion_Air_Fan_Fault_ESV OR Gas_Leak_Check_Switch_Fault_ESV OR Lo_Fire_Limit_Switch_Fault_ESV;
END_PROGRAM

PROGRAM OUTPUT (* task: Scan Program *)
VAR
    ECOR_TRIP : BOOL;
    INST : TOF;
    NO2SHUT : BOOL;
    O502 AT %MW3.0 : BOOL; (* BURNER LOAD UP *)
    O503 AT %MW3.1 : BOOL; (* LOW CIRCULATION FAN SPEED *)
    O504 AT %MW3.2 : BOOL; (* BURNER START *)
    O505 AT %MW3.3 : BOOL;
    O506 AT %MW3.4 : BOOL; (* HIGH TEMPERATURE *)
    O507 AT %MW3.5 : BOOL; (* MISS FIRE *)
    O508 AT %MW3.6 : BOOL; (* HIGH GAS PRESSURE *)
    O509 AT %MW3.7 : BOOL; (* LOW GAS PRESSURE *)
    O510 AT %MW3.8 : BOOL; (* GAS LEAK FAULT *)
    O511 AT %MW3.9 : BOOL; (* PURGE START *)
    O512 AT %MW3.10 : BOOL; (* PURGE END *)
    O513 AT %MW3.11 : BOOL; (* NO 1 LOW COMBUSTION FAN PRESSURE *)
    O514 AT %MW3.12 : BOOL; (* NO 1 LOW COMBUSTION FAN RUNNING *)
    O515 AT %MW3.13 : BOOL; (* NO 2 LOW COMBUSTION FAN PRESSURE *)
    O516 AT %MW3.14 : BOOL; (* NO 2 LOW COMBUSTION FAN RUNNING *)
    O517 AT %MW3.15 : BOOL;
    O518 AT %MW2.14 : BOOL; (* NO.01 COMBUSTION FAN ECOR TRIP *)
    O519 AT %MW2.15 : BOOL; (* NO.02 COMBUSTION FAN ECOR TRIP *)
    OV_1L_1_SHUT_VAL AT %MW2.2 : BOOL; (* 1 MAIN SHUT OFF VALVE *)
    OV_1L_2_SHUT_VAL AT %MW2.3 : BOOL; (* 2 MAIN SHUT -OFF VALVE *)
    OV_1L_PILOT_VAL AT %MW2.1 : BOOL; (* #1 PILOT SOLENOID VALVE *)
    OV_1L_SPK_IGN AT %MW2.0 : BOOL; (* #1 SPARK IGNITOR *)
    OV_1_COMB_FAN_RUN AT %MW2.6 : BOOL; (* #1 COMBUSION AIR FAN RUN *)
    OV_2L_PILOT_VAL AT %MW2.5 : BOOL; (* #2 PILOT SOLENOID VALVE *)
    OV_2L_SPK_IGN AT %MW2.4 : BOOL; (* #2 SPARK IGNITOR *)
    OV_2_COMB_FAN_RUN AT %MW2.7 : BOOL; (* #2 COMBUSION AIR FAN RUN *)
END_VAR

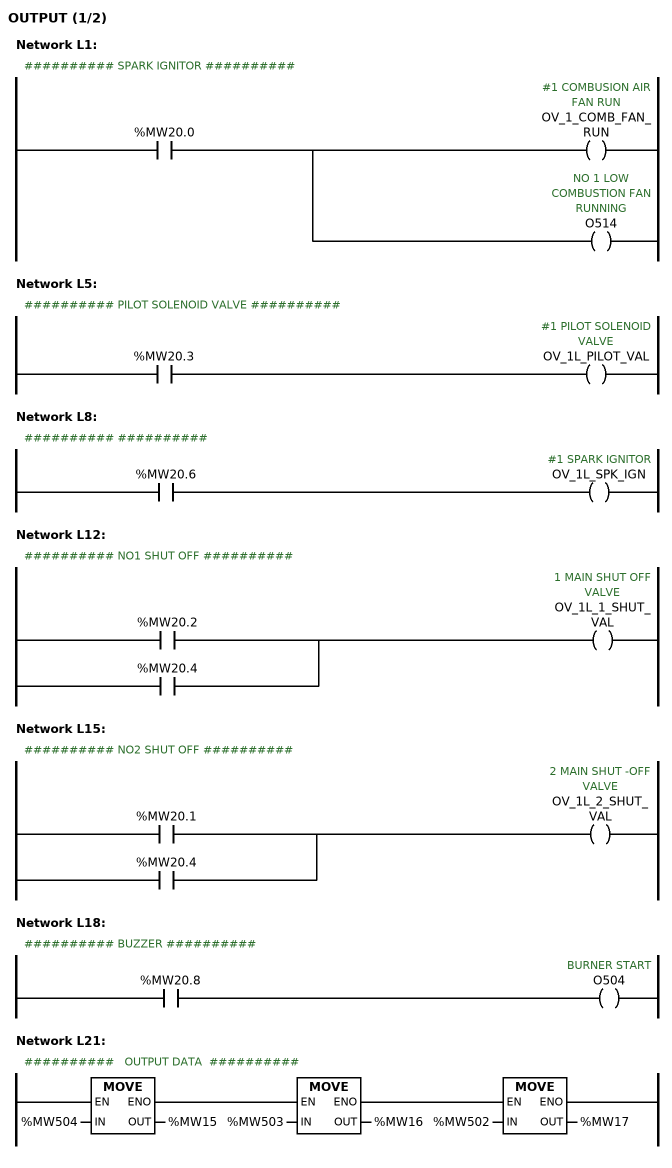
(* ########## SPARK IGNITOR ########## *)
(* Rung L1 *)
OV_1_COMB_FAN_RUN := %MW20.0;
O514 := %MW20.0;
(* ########## PILOT SOLENOID VALVE ########## *)
(* Rung L5 *)
OV_1L_PILOT_VAL := %MW20.3;
(* ########## ########## *)
(* Rung L8 *)
OV_1L_SPK_IGN := %MW20.6;
(* ########## NO1 SHUT OFF ########## *)
(* Rung L12 *)
OV_1L_1_SHUT_VAL := %MW20.2 OR %MW20.4;
(* ########## NO2 SHUT OFF ########## *)
(* Rung L15 *)
OV_1L_2_SHUT_VAL := %MW20.1 OR %MW20.4;
(* ########## BUZZER ########## *)
(* Rung L18 *)
O504 := %MW20.8;
(* ##########   OUTPUT DATA  ########## *)
(* Rung L21 *)
%MW15 := %MW504;
%MW16 := %MW503;
%MW17 := %MW502;

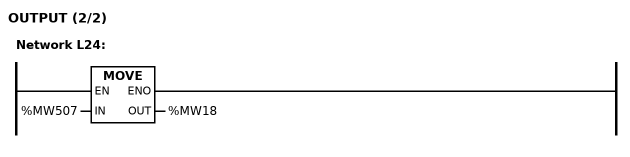
(* Rung L24 *)
%MW18 := %MW507;
END_PROGRAM